// TwinCAT 3 PLC project FMTimeTests
// ProgramVersion: 3.1.4024.0
// libraries:
//   Tc2_Standard, * (Beckhoff Automation GmbH)
//   Tc3_Module, * (Beckhoff Automation GmbH)
//   TcUnit, * (www.tcunit.org)
//   Times, * (TomasRompotl)
// project tree:
//   Clocks/ PeriodicTriggerTest.TcPOU (not stored)
//   Convert/ ConvertFunctionsTest.TcPOU (not stored)
//   / PlcTask.TcTTO (not stored), PRG_Test.TcPOU
// (motion and I/O tree: see PLC project fmtypestests)
// real-time tasks:
//   TASK FMTypesTestsTask: cycle T#1ms, priority 20, ADS port 350
//   TASK FMStringsTestsTask: cycle T#1ms, priority 21, ADS port 351
//   TASK FMDataTestsTask: cycle T#1ms, priority 22, ADS port 352
//   TASK FMMathTestsTask: cycle T#1ms, priority 23, ADS port 353
//   TASK FMTimeTestsTask: cycle T#1ms, priority 24, ADS port 354

// ---- PRG_Test.TcPOU
PROGRAM PRG_Test
VAR
	convertFunctionsTest : ConvertFunctionsTest;
	periodicTriggerTest : PeriodicTriggerTest;
END_VAR

TcUnit.RUN();

END_PROGRAM
